// TIA Portal V16 export
// export: Created 2024-09-05T17:40:13.7980906Z, ExportSetting WithDefaults, DisplayName Totally Integrated Automation Portal, DisplayVersion V16 Update 6, DisplayName TIA Portal Version Control Interface, DisplayVersion V16 Update 2, DisplayName TIA Portal Openness, DisplayVersion V16 Update 6, DisplayName STEP 7 Professional, DisplayVersion V16 Update 6, DisplayName STEP 7 Safety, DisplayVersion V16, DisplayName WinCC Advanced, DisplayVersion V16 Update 6
TYPE "UDT_Digiforce_receive"
// stored: IsFailsafeCompliant false
   STRUCT
      dataD : Struct
         Ready : Bool;
         OK : Bool;
         NOK : Bool;
         NOK_ONL : Bool;
         S1 : Bool;
         S2 : Bool;
         OK_STEST : Bool;
         MEAS_ACT : Bool;
         Strobe : Bool;
         Prog0 : Bool;
         Prog1 : Bool;
         Prog2 : Bool;
         reserve1 : Bool;
         reserve2 : Bool;
         reserve3 : Bool;
         reserve4 : Bool;
         Global_NOK : Bool;
         "Overload _NOK" : Bool;
         Window_1_NOK : Bool;
         Window_2_NOK : Bool;
         Window_3_NOK : Bool;
         Threshold_1_NOK : Bool;
         Threshold_2_NOK : Bool;
         Trapezoid_1_NOK : Bool;
         Trapezoid2_NOK : Bool;
         Envelope_NOK : Bool;
         "Measurement_w/o_READY" : Bool;
         USB_logging_error : Bool;
         reserve5 : Bool;
         reserve6 : Bool;
         reserve7 : Bool;
         reserve8 : Bool;
      END_STRUCT;
      dataA : Array[1..22] of Real;
   END_STRUCT;
END_TYPE
